{attribute 'GeneratedUsingTerminal: EK1122-0000-0018'}
{attribute addProperty BoxType "EK1122-0000-0018"}
{attribute addProperty Id "Beckhoff_ELM35xxsub_EK1100EK1100_1FC0878B2"}
{attribute addProperty CRC "259085035"}
{attribute addProperty Size "2"}
TYPE Beckhoff_ELM35xxEK1122_0F7152EB EXTENDS EK1122_1FC0878B :
STRUCT
	{attribute addProperty Name "Beckhoff ELM35xxsub EK1100"}
	{attribute addProperty PreviousPort "Beckhoff ELM35xxEK1122 : D"}
	Beckhoff_ELM35xxsub_EK1100 : EK1100_1FC0878B;
END_STRUCT
END_TYPE

(* stored: Version 1.2.0.0, ProductVersion 3.1.4024.9
   DUT Beckhoff_ELM35xxEK1122_0F7152EB: Id {d0ae1844-c68e-43d3-bfa6-9eae69d6c348} *)
